(* CODESYS project e!C_OPCUA_Test_1.ecp

Project tree, tasks and I/O mapping:
  PFC200_CS_2ETH_CAN : 750-8203 PFC200 2ETH CAN, WAGO, order no. 0750-8203, version 5.11.1.16
    application Application
      task PLC_Task (cyclic, interval t#10ms, priority 14) calls PLC_PRG
      Symbols
      global variables GVL
      program PLC_PRG [ST]
    DeviceAdapter
    Kbus : Kbus, WAGO, version 1.4.0.2
        unmapped channels: K-BUS diagnostics
      _8_DO_DI_Generic : 075x-8DO8DI, WAGO, order no. 075x-8DO8DI, version 0.0.0.13
          settings: K-BUS Module slot index = 1
          unmapped channels: _IN, _OUT
        DeviceAdapter
    MODBUS
      MODBUS : MODBUS, WAGO, order no. n/a, version 1.1.1.15
    CANbus
*)

// PFC200_CS_2ETH_CAN/Application/GVL
VAR_GLOBAL
	minopcvar1: WORD;
END_VAR

// PFC200_CS_2ETH_CAN/Application/PLC_PRG
PROGRAM PLC_PRG
VAR
END_VAR

minopcvar1;

END_PROGRAM
